SUBAPPLICATION Change_Softkey_Mask (* Subapplication Type *)
  (* Standard: 61499-2 *)
  (* Version 1.0, 2026-01-24, 04jul *)
  IMPORT logiBUS::io::DI::logiBUS_DI::Input_I1;
  IMPORT logiBUS::io::DQ::logiBUS_DO::Output_Q1;
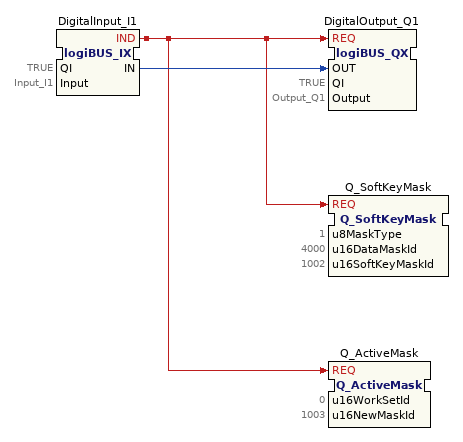
  FBS
    DigitalOutput_Q1 : logiBUS::io::DQ::logiBUS_QX(QI := TRUE, Output := Output_Q1);
    DigitalInput_I1 : logiBUS::io::DI::logiBUS_IX(QI := TRUE, Input := Input_I1);
    Q_SoftKeyMask : isobus::UT::Q::Q_SoftKeyMask(u8MaskType := 1, u16DataMaskId := 4000, u16SoftKeyMaskId := 1002);
    Q_ActiveMask : isobus::UT::Q::Q_ActiveMask(u16WorkSetId := 0, u16NewMaskId := 1003);
  END_FBS
  EVENT_CONNECTIONS
    DigitalInput_I1.IND TO DigitalOutput_Q1.REQ;
    DigitalInput_I1.IND TO Q_SoftKeyMask.REQ;
    DigitalInput_I1.IND TO Q_ActiveMask.REQ;
  END_CONNECTIONS
  DATA_CONNECTIONS
    DigitalInput_I1.IN TO DigitalOutput_Q1.OUT;
  END_CONNECTIONS
END_SUBAPPLICATION
